aff1C[0  , 0] := 1.00000E+01; aff1C[0  , 1] := -4.03481E+00;
aff1C[1  , 0] := 1.99800E+01; aff1C[1  , 1] := -3.16200E+00;
aff1C[2  , 0] := 2.99600E+01; aff1C[2  , 1] := -2.64479E+00;
aff1C[3  , 0] := 3.99400E+01; aff1C[3  , 1] := -2.31488E+00;
aff1C[4  , 0] := 4.99200E+01; aff1C[4  , 1] := -2.09732E+00;
aff1C[5  , 0] := 5.99000E+01; aff1C[5  , 1] := -1.95840E+00;
aff1C[6  , 0] := 6.98800E+01; aff1C[6  , 1] := -1.87113E+00;
aff1C[7  , 0] := 7.98600E+01; aff1C[7  , 1] := -1.81732E+00;
aff1C[8  , 0] := 8.98400E+01; aff1C[8  , 1] := -1.78617E+00;
aff1C[9  , 0] := 9.98200E+01; aff1C[9  , 1] := -1.77164E+00;
aff1C[10 , 0] := 1.09800E+02; aff1C[10 , 1] := -1.76959E+00;
aff1C[11 , 0] := 1.19780E+02; aff1C[11 , 1] := -1.77729E+00;
aff1C[12 , 0] := 1.29760E+02; aff1C[12 , 1] := -1.79375E+00;
aff1C[13 , 0] := 1.39740E+02; aff1C[13 , 1] := -1.81862E+00;
aff1C[14 , 0] := 1.49720E+02; aff1C[14 , 1] := -1.85102E+00;
aff1C[15 , 0] := 1.59700E+02; aff1C[15 , 1] := -1.89079E+00;
aff1C[16 , 0] := 1.69680E+02; aff1C[16 , 1] := -1.93825E+00;
aff1C[17 , 0] := 1.79660E+02; aff1C[17 , 1] := -1.99421E+00;
aff1C[18 , 0] := 1.89640E+02; aff1C[18 , 1] := -2.05996E+00;
aff1C[19 , 0] := 1.99620E+02; aff1C[19 , 1] := -2.13743E+00;
aff1C[20 , 0] := 2.09600E+02; aff1C[20 , 1] := -2.22948E+00;
aff1C[21 , 0] := 2.19580E+02; aff1C[21 , 1] := -2.34037E+00;
aff1C[22 , 0] := 2.29560E+02; aff1C[22 , 1] := -2.47673E+00;
aff1C[23 , 0] := 2.39540E+02; aff1C[23 , 1] := -2.64947E+00;
aff1C[24 , 0] := 2.49520E+02; aff1C[24 , 1] := -2.87833E+00;
aff1C[25 , 0] := 2.59500E+02; aff1C[25 , 1] := -3.20451E+00;
aff1C[26 , 0] := 2.69480E+02; aff1C[26 , 1] := -3.73879E+00;
aff1C[27 , 0] := 2.79460E+02; aff1C[27 , 1] := -5.04188E+00;
aff1C[28 , 0] := 2.89440E+02; aff1C[28 , 1] := -4.53653E+00;
aff1C[29 , 0] := 2.99420E+02; aff1C[29 , 1] := -3.20323E+00;
aff1C[30 , 0] := 3.09400E+02; aff1C[30 , 1] := -2.53148E+00;
aff1C[31 , 0] := 3.19380E+02; aff1C[31 , 1] := -2.07370E+00;
aff1C[32 , 0] := 3.29360E+02; aff1C[32 , 1] := -1.72635E+00;
aff1C[33 , 0] := 3.39340E+02; aff1C[33 , 1] := -1.44913E+00;
aff1C[34 , 0] := 3.49320E+02; aff1C[34 , 1] := -1.22093E+00;
aff1C[35 , 0] := 3.59300E+02; aff1C[35 , 1] := -1.02921E+00;
aff1C[36 , 0] := 3.69280E+02; aff1C[36 , 1] := -8.65802E-01;
aff1C[37 , 0] := 3.79260E+02; aff1C[37 , 1] := -7.25116E-01;
aff1C[38 , 0] := 3.89240E+02; aff1C[38 , 1] := -6.03050E-01;
aff1C[39 , 0] := 3.99220E+02; aff1C[39 , 1] := -4.96466E-01;
aff1C[40 , 0] := 4.09200E+02; aff1C[40 , 1] := -4.02926E-01;
aff1C[41 , 0] := 4.19180E+02; aff1C[41 , 1] := -3.20489E-01;
aff1C[42 , 0] := 4.29160E+02; aff1C[42 , 1] := -2.47581E-01;
aff1C[43 , 0] := 4.39140E+02; aff1C[43 , 1] := -1.82911E-01;
aff1C[44 , 0] := 4.49120E+02; aff1C[44 , 1] := -1.25405E-01;
aff1C[45 , 0] := 4.59100E+02; aff1C[45 , 1] := -7.41593E-02;
aff1C[46 , 0] := 4.69080E+02; aff1C[46 , 1] := -2.84093E-02;
aff1C[47 , 0] := 4.79060E+02; aff1C[47 , 1] := 1.24973E-02;
aff1C[48 , 0] := 4.89040E+02; aff1C[48 , 1] := 4.91208E-02;
aff1C[49 , 0] := 4.99020E+02; aff1C[49 , 1] := 8.19448E-02;
aff1C[50 , 0] := 5.09000E+02; aff1C[50 , 1] := 1.11389E-01;
aff1C[51 , 0] := 5.18980E+02; aff1C[51 , 1] := 1.37819E-01;
aff1C[52 , 0] := 5.28960E+02; aff1C[52 , 1] := 1.61554E-01;
aff1C[53 , 0] := 5.38940E+02; aff1C[53 , 1] := 1.82875E-01;
aff1C[54 , 0] := 5.48920E+02; aff1C[54 , 1] := 2.02029E-01;
aff1C[55 , 0] := 5.58900E+02; aff1C[55 , 1] := 2.19234E-01;
aff1C[56 , 0] := 5.68880E+02; aff1C[56 , 1] := 2.34684E-01;
aff1C[57 , 0] := 5.78860E+02; aff1C[57 , 1] := 2.48550E-01;
aff1C[58 , 0] := 5.88840E+02; aff1C[58 , 1] := 2.60984E-01;
aff1C[59 , 0] := 5.98820E+02; aff1C[59 , 1] := 2.72123E-01;
aff1C[60 , 0] := 6.08800E+02; aff1C[60 , 1] := 2.82088E-01;
aff1C[61 , 0] := 6.18780E+02; aff1C[61 , 1] := 2.90989E-01;
aff1C[62 , 0] := 6.28760E+02; aff1C[62 , 1] := 2.98923E-01;
aff1C[63 , 0] := 6.38740E+02; aff1C[63 , 1] := 3.05978E-01;
aff1C[64 , 0] := 6.48720E+02; aff1C[64 , 1] := 3.12234E-01;
aff1C[65 , 0] := 6.58700E+02; aff1C[65 , 1] := 3.17761E-01;
aff1C[66 , 0] := 6.68680E+02; aff1C[66 , 1] := 3.22624E-01;
aff1C[67 , 0] := 6.78660E+02; aff1C[67 , 1] := 3.26882E-01;
aff1C[68 , 0] := 6.88640E+02; aff1C[68 , 1] := 3.30587E-01;
aff1C[69 , 0] := 6.98620E+02; aff1C[69 , 1] := 3.33787E-01;
aff1C[70 , 0] := 7.08600E+02; aff1C[70 , 1] := 3.36525E-01;
aff1C[71 , 0] := 7.18580E+02; aff1C[71 , 1] := 3.38842E-01;
aff1C[72 , 0] := 7.28560E+02; aff1C[72 , 1] := 3.40773E-01;
aff1C[73 , 0] := 7.38540E+02; aff1C[73 , 1] := 3.42351E-01;
aff1C[74 , 0] := 7.48520E+02; aff1C[74 , 1] := 3.43606E-01;
aff1C[75 , 0] := 7.58500E+02; aff1C[75 , 1] := 3.44565E-01;
aff1C[76 , 0] := 7.68480E+02; aff1C[76 , 1] := 3.45254E-01;
aff1C[77 , 0] := 7.78460E+02; aff1C[77 , 1] := 3.45694E-01;
aff1C[78 , 0] := 7.88440E+02; aff1C[78 , 1] := 3.45908E-01;
aff1C[79 , 0] := 7.98420E+02; aff1C[79 , 1] := 3.45914E-01;
aff1C[80 , 0] := 8.08400E+02; aff1C[80 , 1] := 3.45729E-01;
aff1C[81 , 0] := 8.18380E+02; aff1C[81 , 1] := 3.45371E-01;
aff1C[82 , 0] := 8.28360E+02; aff1C[82 , 1] := 3.44854E-01;
aff1C[83 , 0] := 8.38340E+02; aff1C[83 , 1] := 3.44196E-01;
aff1C[84 , 0] := 8.48320E+02; aff1C[84 , 1] := 3.43361E-01;
aff1C[85 , 0] := 8.58300E+02; aff1C[85 , 1] := 3.42839E-01;
aff1C[86 , 0] := 8.68280E+02; aff1C[86 , 1] := 3.41862E-01;
aff1C[87 , 0] := 8.78260E+02; aff1C[87 , 1] := 3.40748E-01;
aff1C[88 , 0] := 8.88240E+02; aff1C[88 , 1] := 3.39538E-01;
aff1C[89 , 0] := 8.98220E+02; aff1C[89 , 1] := 3.38248E-01;
aff1C[90 , 0] := 9.08200E+02; aff1C[90 , 1] := 3.36883E-01;
aff1C[91 , 0] := 9.18180E+02; aff1C[91 , 1] := 3.35451E-01;
aff1C[92 , 0] := 9.28160E+02; aff1C[92 , 1] := 3.33958E-01;
aff1C[93 , 0] := 9.38140E+02; aff1C[93 , 1] := 3.32411E-01;
aff1C[94 , 0] := 9.48120E+02; aff1C[94 , 1] := 3.30816E-01;
aff1C[95 , 0] := 9.58100E+02; aff1C[95 , 1] := 3.29178E-01;
aff1C[96 , 0] := 9.68080E+02; aff1C[96 , 1] := 3.27503E-01;
aff1C[97 , 0] := 9.78060E+02; aff1C[97 , 1] := 3.25794E-01;
aff1C[98 , 0] := 9.88040E+02; aff1C[98 , 1] := 3.24057E-01;
aff1C[99 , 0] := 9.98020E+02; aff1C[99 , 1] := 3.22295E-01;
aff1C[100, 0] := 1.00800E+03; aff1C[100, 1] := 3.20475E-01;
aff1C[101, 0] := 1.01798E+03; aff1C[101, 1] := 3.18626E-01;
aff1C[102, 0] := 1.02796E+03; aff1C[102, 1] := 3.16761E-01;
aff1C[103, 0] := 1.03794E+03; aff1C[103, 1] := 3.14881E-01;
aff1C[104, 0] := 1.04792E+03; aff1C[104, 1] := 3.12989E-01;
aff1C[105, 0] := 1.05790E+03; aff1C[105, 1] := 3.11086E-01;
aff1C[106, 0] := 1.06788E+03; aff1C[106, 1] := 3.09176E-01;
aff1C[107, 0] := 1.07786E+03; aff1C[107, 1] := 3.07262E-01;
aff1C[108, 0] := 1.08784E+03; aff1C[108, 1] := 3.05346E-01;
aff1C[109, 0] := 1.09782E+03; aff1C[109, 1] := 3.03433E-01;
aff1C[110, 0] := 1.10780E+03; aff1C[110, 1] := 3.01524E-01;
aff1C[111, 0] := 1.11778E+03; aff1C[111, 1] := 2.99623E-01;
aff1C[112, 0] := 1.12776E+03; aff1C[112, 1] := 2.97736E-01;
aff1C[113, 0] := 1.13774E+03; aff1C[113, 1] := 2.95857E-01;
aff1C[114, 0] := 1.14772E+03; aff1C[114, 1] := 2.93954E-01;
aff1C[115, 0] := 1.15770E+03; aff1C[115, 1] := 2.92011E-01;
aff1C[116, 0] := 1.16768E+03; aff1C[116, 1] := 2.90036E-01;
aff1C[117, 0] := 1.17766E+03; aff1C[117, 1] := 2.88036E-01;
aff1C[118, 0] := 1.18764E+03; aff1C[118, 1] := 2.86016E-01;
aff1C[119, 0] := 1.19762E+03; aff1C[119, 1] := 2.83981E-01;
aff1C[120, 0] := 1.20760E+03; aff1C[120, 1] := 2.81934E-01;
aff1C[121, 0] := 1.21758E+03; aff1C[121, 1] := 2.79880E-01;
aff1C[122, 0] := 1.22756E+03; aff1C[122, 1] := 2.77820E-01;
aff1C[123, 0] := 1.23754E+03; aff1C[123, 1] := 2.75758E-01;
aff1C[124, 0] := 1.24752E+03; aff1C[124, 1] := 2.73697E-01;
aff1C[125, 0] := 1.25750E+03; aff1C[125, 1] := 2.71637E-01;
aff1C[126, 0] := 1.26748E+03; aff1C[126, 1] := 2.69581E-01;
aff1C[127, 0] := 1.27746E+03; aff1C[127, 1] := 2.67530E-01;
aff1C[128, 0] := 1.28744E+03; aff1C[128, 1] := 2.65487E-01;
aff1C[129, 0] := 1.29742E+03; aff1C[129, 1] := 2.63451E-01;
aff1C[130, 0] := 1.30740E+03; aff1C[130, 1] := 2.61425E-01;
aff1C[131, 0] := 1.31738E+03; aff1C[131, 1] := 2.59409E-01;
aff1C[132, 0] := 1.32736E+03; aff1C[132, 1] := 2.57404E-01;
aff1C[133, 0] := 1.33734E+03; aff1C[133, 1] := 2.55410E-01;
aff1C[134, 0] := 1.34732E+03; aff1C[134, 1] := 2.53430E-01;
aff1C[135, 0] := 1.35730E+03; aff1C[135, 1] := 2.51462E-01;
aff1C[136, 0] := 1.36728E+03; aff1C[136, 1] := 2.49508E-01;
aff1C[137, 0] := 1.37726E+03; aff1C[137, 1] := 2.47568E-01;
aff1C[138, 0] := 1.38724E+03; aff1C[138, 1] := 2.45643E-01;
aff1C[139, 0] := 1.39722E+03; aff1C[139, 1] := 2.43732E-01;
aff1C[140, 0] := 1.40720E+03; aff1C[140, 1] := 2.41837E-01;
aff1C[141, 0] := 1.41718E+03; aff1C[141, 1] := 2.39957E-01;
aff1C[142, 0] := 1.42716E+03; aff1C[142, 1] := 2.38093E-01;
aff1C[143, 0] := 1.43714E+03; aff1C[143, 1] := 2.36244E-01;
aff1C[144, 0] := 1.44712E+03; aff1C[144, 1] := 2.34412E-01;
aff1C[145, 0] := 1.45710E+03; aff1C[145, 1] := 2.32596E-01;
aff1C[146, 0] := 1.46708E+03; aff1C[146, 1] := 2.30796E-01;
aff1C[147, 0] := 1.47706E+03; aff1C[147, 1] := 2.29012E-01;
aff1C[148, 0] := 1.48704E+03; aff1C[148, 1] := 2.27245E-01;
aff1C[149, 0] := 1.49702E+03; aff1C[149, 1] := 2.25494E-01;
aff1C[150, 0] := 1.50700E+03; aff1C[150, 1] := 2.23759E-01;
aff1C[151, 0] := 1.51698E+03; aff1C[151, 1] := 2.22041E-01;
aff1C[152, 0] := 1.52696E+03; aff1C[152, 1] := 2.20340E-01;
aff1C[153, 0] := 1.53694E+03; aff1C[153, 1] := 2.18655E-01;
aff1C[154, 0] := 1.54692E+03; aff1C[154, 1] := 2.16986E-01;
aff1C[155, 0] := 1.55690E+03; aff1C[155, 1] := 2.15333E-01;
aff1C[156, 0] := 1.56688E+03; aff1C[156, 1] := 2.13697E-01;
aff1C[157, 0] := 1.57686E+03; aff1C[157, 1] := 2.12077E-01;
aff1C[158, 0] := 1.58684E+03; aff1C[158, 1] := 2.10473E-01;
aff1C[159, 0] := 1.59682E+03; aff1C[159, 1] := 2.08884E-01;
aff1C[160, 0] := 1.60680E+03; aff1C[160, 1] := 2.07312E-01;
aff1C[161, 0] := 1.61678E+03; aff1C[161, 1] := 2.05756E-01;
aff1C[162, 0] := 1.62676E+03; aff1C[162, 1] := 2.04215E-01;
aff1C[163, 0] := 1.63674E+03; aff1C[163, 1] := 2.02690E-01;
aff1C[164, 0] := 1.64672E+03; aff1C[164, 1] := 2.01180E-01;
aff1C[165, 0] := 1.65670E+03; aff1C[165, 1] := 1.99686E-01;
aff1C[166, 0] := 1.66668E+03; aff1C[166, 1] := 1.98206E-01;
aff1C[167, 0] := 1.67666E+03; aff1C[167, 1] := 1.96742E-01;
aff1C[168, 0] := 1.68664E+03; aff1C[168, 1] := 1.95293E-01;
aff1C[169, 0] := 1.69662E+03; aff1C[169, 1] := 1.93859E-01;
aff1C[170, 0] := 1.70660E+03; aff1C[170, 1] := 1.92439E-01;
aff1C[171, 0] := 1.71658E+03; aff1C[171, 1] := 1.91034E-01;
aff1C[172, 0] := 1.72656E+03; aff1C[172, 1] := 1.89643E-01;
aff1C[173, 0] := 1.73654E+03; aff1C[173, 1] := 1.88266E-01;
aff1C[174, 0] := 1.74652E+03; aff1C[174, 1] := 1.86904E-01;
aff1C[175, 0] := 1.75650E+03; aff1C[175, 1] := 1.85555E-01;
aff1C[176, 0] := 1.76648E+03; aff1C[176, 1] := 1.84221E-01;
aff1C[177, 0] := 1.77646E+03; aff1C[177, 1] := 1.82900E-01;
aff1C[178, 0] := 1.78644E+03; aff1C[178, 1] := 1.81592E-01;
aff1C[179, 0] := 1.79642E+03; aff1C[179, 1] := 1.80298E-01;
aff1C[180, 0] := 1.80640E+03; aff1C[180, 1] := 1.79018E-01;
aff1C[181, 0] := 1.81638E+03; aff1C[181, 1] := 1.77750E-01;
aff1C[182, 0] := 1.82636E+03; aff1C[182, 1] := 1.76495E-01;
aff1C[183, 0] := 1.83634E+03; aff1C[183, 1] := 1.75254E-01;
aff1C[184, 0] := 1.84632E+03; aff1C[184, 1] := 1.74024E-01;
aff1C[185, 0] := 1.85630E+03; aff1C[185, 1] := 1.72808E-01;
aff1C[186, 0] := 1.86628E+03; aff1C[186, 1] := 1.71604E-01;
aff1C[187, 0] := 1.87626E+03; aff1C[187, 1] := 1.70412E-01;
aff1C[188, 0] := 1.88624E+03; aff1C[188, 1] := 1.69232E-01;
aff1C[189, 0] := 1.89622E+03; aff1C[189, 1] := 1.68064E-01;
aff1C[190, 0] := 1.90620E+03; aff1C[190, 1] := 1.66908E-01;
aff1C[191, 0] := 1.91618E+03; aff1C[191, 1] := 1.65764E-01;
aff1C[192, 0] := 1.92616E+03; aff1C[192, 1] := 1.64631E-01;
aff1C[193, 0] := 1.93614E+03; aff1C[193, 1] := 1.63510E-01;
aff1C[194, 0] := 1.94612E+03; aff1C[194, 1] := 1.62400E-01;
aff1C[195, 0] := 1.95610E+03; aff1C[195, 1] := 1.61301E-01;
aff1C[196, 0] := 1.96608E+03; aff1C[196, 1] := 1.60214E-01;
aff1C[197, 0] := 1.97606E+03; aff1C[197, 1] := 1.59137E-01;
aff1C[198, 0] := 1.98604E+03; aff1C[198, 1] := 1.58071E-01;
aff1C[199, 0] := 1.99602E+03; aff1C[199, 1] := 1.57015E-01;
aff1C[200, 0] := 2.00600E+03; aff1C[200, 1] := 1.55971E-01;
aff1C[201, 0] := 2.01598E+03; aff1C[201, 1] := 1.54936E-01;
aff1C[202, 0] := 2.02596E+03; aff1C[202, 1] := 1.53912E-01;
aff1C[203, 0] := 2.03594E+03; aff1C[203, 1] := 1.52898E-01;
aff1C[204, 0] := 2.04592E+03; aff1C[204, 1] := 1.51894E-01;
aff1C[205, 0] := 2.05590E+03; aff1C[205, 1] := 1.50900E-01;
aff1C[206, 0] := 2.06588E+03; aff1C[206, 1] := 1.49916E-01;
aff1C[207, 0] := 2.07586E+03; aff1C[207, 1] := 1.48942E-01;
aff1C[208, 0] := 2.08584E+03; aff1C[208, 1] := 1.47977E-01;
aff1C[209, 0] := 2.09582E+03; aff1C[209, 1] := 1.47022E-01;
aff1C[210, 0] := 2.10580E+03; aff1C[210, 1] := 1.46076E-01;
aff1C[211, 0] := 2.11578E+03; aff1C[211, 1] := 1.45139E-01;
aff1C[212, 0] := 2.12576E+03; aff1C[212, 1] := 1.44211E-01;
aff1C[213, 0] := 2.13574E+03; aff1C[213, 1] := 1.43292E-01;
aff1C[214, 0] := 2.14572E+03; aff1C[214, 1] := 1.42383E-01;
aff1C[215, 0] := 2.15570E+03; aff1C[215, 1] := 1.41482E-01;
aff1C[216, 0] := 2.16568E+03; aff1C[216, 1] := 1.40590E-01;
aff1C[217, 0] := 2.17566E+03; aff1C[217, 1] := 1.39706E-01;
aff1C[218, 0] := 2.18564E+03; aff1C[218, 1] := 1.38831E-01;
aff1C[219, 0] := 2.19562E+03; aff1C[219, 1] := 1.37964E-01;
aff1C[220, 0] := 2.20560E+03; aff1C[220, 1] := 1.37106E-01;
aff1C[221, 0] := 2.21558E+03; aff1C[221, 1] := 1.36256E-01;
aff1C[222, 0] := 2.22556E+03; aff1C[222, 1] := 1.35414E-01;
aff1C[223, 0] := 2.23554E+03; aff1C[223, 1] := 1.34580E-01;
aff1C[224, 0] := 2.24552E+03; aff1C[224, 1] := 1.33753E-01;
aff1C[225, 0] := 2.25550E+03; aff1C[225, 1] := 1.32935E-01;
aff1C[226, 0] := 2.26548E+03; aff1C[226, 1] := 1.32125E-01;
aff1C[227, 0] := 2.27546E+03; aff1C[227, 1] := 1.31322E-01;
aff1C[228, 0] := 2.28544E+03; aff1C[228, 1] := 1.30526E-01;
aff1C[229, 0] := 2.29542E+03; aff1C[229, 1] := 1.29739E-01;
aff1C[230, 0] := 2.30540E+03; aff1C[230, 1] := 1.28958E-01;
aff1C[231, 0] := 2.31538E+03; aff1C[231, 1] := 1.28185E-01;
aff1C[232, 0] := 2.32536E+03; aff1C[232, 1] := 1.27419E-01;
aff1C[233, 0] := 2.33534E+03; aff1C[233, 1] := 1.26660E-01;
aff1C[234, 0] := 2.34532E+03; aff1C[234, 1] := 1.25908E-01;
aff1C[235, 0] := 2.35530E+03; aff1C[235, 1] := 1.25164E-01;
aff1C[236, 0] := 2.36528E+03; aff1C[236, 1] := 1.24426E-01;
aff1C[237, 0] := 2.37526E+03; aff1C[237, 1] := 1.23695E-01;
aff1C[238, 0] := 2.38524E+03; aff1C[238, 1] := 1.22970E-01;
aff1C[239, 0] := 2.39522E+03; aff1C[239, 1] := 1.22253E-01;
aff1C[240, 0] := 2.40520E+03; aff1C[240, 1] := 1.21541E-01;
aff1C[241, 0] := 2.41518E+03; aff1C[241, 1] := 1.20837E-01;
aff1C[242, 0] := 2.42516E+03; aff1C[242, 1] := 1.20139E-01;
aff1C[243, 0] := 2.43514E+03; aff1C[243, 1] := 1.19447E-01;
aff1C[244, 0] := 2.44512E+03; aff1C[244, 1] := 1.18761E-01;
aff1C[245, 0] := 2.45510E+03; aff1C[245, 1] := 1.18082E-01;
aff1C[246, 0] := 2.46508E+03; aff1C[246, 1] := 1.17409E-01;
aff1C[247, 0] := 2.47506E+03; aff1C[247, 1] := 1.16742E-01;
aff1C[248, 0] := 2.48504E+03; aff1C[248, 1] := 1.16081E-01;
aff1C[249, 0] := 2.49502E+03; aff1C[249, 1] := 1.15426E-01;
aff1C[250, 0] := 2.50500E+03; aff1C[250, 1] := 1.14777E-01;
aff1C[251, 0] := 2.51498E+03; aff1C[251, 1] := 1.14134E-01;
aff1C[252, 0] := 2.52496E+03; aff1C[252, 1] := 1.13496E-01;
aff1C[253, 0] := 2.53494E+03; aff1C[253, 1] := 1.12864E-01;
aff1C[254, 0] := 2.54492E+03; aff1C[254, 1] := 1.12238E-01;
aff1C[255, 0] := 2.55490E+03; aff1C[255, 1] := 1.11617E-01;
aff1C[256, 0] := 2.56488E+03; aff1C[256, 1] := 1.11002E-01;
aff1C[257, 0] := 2.57486E+03; aff1C[257, 1] := 1.10393E-01;
aff1C[258, 0] := 2.58484E+03; aff1C[258, 1] := 1.09789E-01;
aff1C[259, 0] := 2.59482E+03; aff1C[259, 1] := 1.09190E-01;
aff1C[260, 0] := 2.60480E+03; aff1C[260, 1] := 1.08596E-01;
aff1C[261, 0] := 2.61478E+03; aff1C[261, 1] := 1.08008E-01;
aff1C[262, 0] := 2.62476E+03; aff1C[262, 1] := 1.07425E-01;
aff1C[263, 0] := 2.63474E+03; aff1C[263, 1] := 1.06847E-01;
aff1C[264, 0] := 2.64472E+03; aff1C[264, 1] := 1.06274E-01;
aff1C[265, 0] := 2.65470E+03; aff1C[265, 1] := 1.05706E-01;
aff1C[266, 0] := 2.66468E+03; aff1C[266, 1] := 1.05143E-01;
aff1C[267, 0] := 2.67466E+03; aff1C[267, 1] := 1.04585E-01;
aff1C[268, 0] := 2.68464E+03; aff1C[268, 1] := 1.04032E-01;
aff1C[269, 0] := 2.69462E+03; aff1C[269, 1] := 1.03484E-01;
aff1C[270, 0] := 2.70460E+03; aff1C[270, 1] := 1.02940E-01;
aff1C[271, 0] := 2.71458E+03; aff1C[271, 1] := 1.02402E-01;
aff1C[272, 0] := 2.72456E+03; aff1C[272, 1] := 1.01868E-01;
aff1C[273, 0] := 2.73454E+03; aff1C[273, 1] := 1.01338E-01;
aff1C[274, 0] := 2.74452E+03; aff1C[274, 1] := 1.00813E-01;
aff1C[275, 0] := 2.75450E+03; aff1C[275, 1] := 1.00293E-01;
aff1C[276, 0] := 2.76448E+03; aff1C[276, 1] := 9.97774E-02;
aff1C[277, 0] := 2.77446E+03; aff1C[277, 1] := 9.92662E-02;
aff1C[278, 0] := 2.78444E+03; aff1C[278, 1] := 9.87594E-02;
aff1C[279, 0] := 2.79442E+03; aff1C[279, 1] := 9.82570E-02;
aff1C[280, 0] := 2.80440E+03; aff1C[280, 1] := 9.77590E-02;
aff1C[281, 0] := 2.81438E+03; aff1C[281, 1] := 9.72652E-02;
aff1C[282, 0] := 2.82436E+03; aff1C[282, 1] := 9.67758E-02;
aff1C[283, 0] := 2.83434E+03; aff1C[283, 1] := 9.62906E-02;
aff1C[284, 0] := 2.84432E+03; aff1C[284, 1] := 9.58096E-02;
aff1C[285, 0] := 2.85430E+03; aff1C[285, 1] := 9.53328E-02;
aff1C[286, 0] := 2.86428E+03; aff1C[286, 1] := 9.48602E-02;
aff1C[287, 0] := 2.87426E+03; aff1C[287, 1] := 9.43916E-02;
aff1C[288, 0] := 2.88424E+03; aff1C[288, 1] := 9.39271E-02;
aff1C[289, 0] := 2.89422E+03; aff1C[289, 1] := 9.34666E-02;
aff1C[290, 0] := 2.90420E+03; aff1C[290, 1] := 9.30102E-02;
aff1C[291, 0] := 2.91418E+03; aff1C[291, 1] := 9.25577E-02;
aff1C[292, 0] := 2.92416E+03; aff1C[292, 1] := 9.21092E-02;
aff1C[293, 0] := 2.93414E+03; aff1C[293, 1] := 9.16645E-02;
aff1C[294, 0] := 2.94412E+03; aff1C[294, 1] := 9.12237E-02;
aff1C[295, 0] := 2.95410E+03; aff1C[295, 1] := 9.07871E-02;
aff1C[296, 0] := 2.96408E+03; aff1C[296, 1] := 9.03545E-02;
aff1C[297, 0] := 2.97406E+03; aff1C[297, 1] := 8.99253E-02;
aff1C[298, 0] := 2.98404E+03; aff1C[298, 1] := 8.94991E-02;
aff1C[299, 0] := 2.99402E+03; aff1C[299, 1] := 8.90753E-02;
aff1C[300, 0] := 3.00400E+03; aff1C[300, 1] := 8.86529E-02;
aff1C[301, 0] := 3.01398E+03; aff1C[301, 1] := 8.82307E-02;
aff1C[302, 0] := 3.02396E+03; aff1C[302, 1] := 8.78083E-02;
aff1C[303, 0] := 3.03394E+03; aff1C[303, 1] := 8.73870E-02;
aff1C[304, 0] := 3.04392E+03; aff1C[304, 1] := 8.69680E-02;
aff1C[305, 0] := 3.05390E+03; aff1C[305, 1] := 8.65522E-02;
aff1C[306, 0] := 3.06388E+03; aff1C[306, 1] := 8.61393E-02;
aff1C[307, 0] := 3.07386E+03; aff1C[307, 1] := 8.57290E-02;
aff1C[308, 0] := 3.08384E+03; aff1C[308, 1] := 8.53210E-02;
aff1C[309, 0] := 3.09382E+03; aff1C[309, 1] := 8.49154E-02;
aff1C[310, 0] := 3.10380E+03; aff1C[310, 1] := 8.45123E-02;
aff1C[311, 0] := 3.11378E+03; aff1C[311, 1] := 8.41118E-02;
aff1C[312, 0] := 3.12376E+03; aff1C[312, 1] := 8.37137E-02;
aff1C[313, 0] := 3.13374E+03; aff1C[313, 1] := 8.33180E-02;
aff1C[314, 0] := 3.14372E+03; aff1C[314, 1] := 8.29248E-02;
aff1C[315, 0] := 3.15370E+03; aff1C[315, 1] := 8.25341E-02;
aff1C[316, 0] := 3.16368E+03; aff1C[316, 1] := 8.21458E-02;
aff1C[317, 0] := 3.17366E+03; aff1C[317, 1] := 8.17599E-02;
aff1C[318, 0] := 3.18364E+03; aff1C[318, 1] := 8.13764E-02;
aff1C[319, 0] := 3.19362E+03; aff1C[319, 1] := 8.09953E-02;
aff1C[320, 0] := 3.20360E+03; aff1C[320, 1] := 8.06166E-02;
aff1C[321, 0] := 3.21358E+03; aff1C[321, 1] := 8.02403E-02;
aff1C[322, 0] := 3.22356E+03; aff1C[322, 1] := 7.98663E-02;
aff1C[323, 0] := 3.23354E+03; aff1C[323, 1] := 7.94947E-02;
aff1C[324, 0] := 3.24352E+03; aff1C[324, 1] := 7.91254E-02;
aff1C[325, 0] := 3.25350E+03; aff1C[325, 1] := 7.87584E-02;
aff1C[326, 0] := 3.26348E+03; aff1C[326, 1] := 7.83938E-02;
aff1C[327, 0] := 3.27346E+03; aff1C[327, 1] := 7.80314E-02;
aff1C[328, 0] := 3.28344E+03; aff1C[328, 1] := 7.76714E-02;
aff1C[329, 0] := 3.29342E+03; aff1C[329, 1] := 7.73136E-02;
aff1C[330, 0] := 3.30340E+03; aff1C[330, 1] := 7.69580E-02;
aff1C[331, 0] := 3.31338E+03; aff1C[331, 1] := 7.66047E-02;
aff1C[332, 0] := 3.32336E+03; aff1C[332, 1] := 7.62536E-02;
aff1C[333, 0] := 3.33334E+03; aff1C[333, 1] := 7.59048E-02;
aff1C[334, 0] := 3.34332E+03; aff1C[334, 1] := 7.55581E-02;
aff1C[335, 0] := 3.35330E+03; aff1C[335, 1] := 7.52136E-02;
aff1C[336, 0] := 3.36328E+03; aff1C[336, 1] := 7.48713E-02;
aff1C[337, 0] := 3.37326E+03; aff1C[337, 1] := 7.45311E-02;
aff1C[338, 0] := 3.38324E+03; aff1C[338, 1] := 7.41931E-02;
aff1C[339, 0] := 3.39322E+03; aff1C[339, 1] := 7.38572E-02;
aff1C[340, 0] := 3.40320E+03; aff1C[340, 1] := 7.35234E-02;
aff1C[341, 0] := 3.41318E+03; aff1C[341, 1] := 7.31918E-02;
aff1C[342, 0] := 3.42316E+03; aff1C[342, 1] := 7.28622E-02;
aff1C[343, 0] := 3.43314E+03; aff1C[343, 1] := 7.25346E-02;
aff1C[344, 0] := 3.44312E+03; aff1C[344, 1] := 7.22092E-02;
aff1C[345, 0] := 3.45310E+03; aff1C[345, 1] := 7.18857E-02;
aff1C[346, 0] := 3.46308E+03; aff1C[346, 1] := 7.15643E-02;
aff1C[347, 0] := 3.47306E+03; aff1C[347, 1] := 7.12450E-02;
aff1C[348, 0] := 3.48304E+03; aff1C[348, 1] := 7.09276E-02;
aff1C[349, 0] := 3.49302E+03; aff1C[349, 1] := 7.06122E-02;
aff1C[350, 0] := 3.50300E+03; aff1C[350, 1] := 7.02987E-02;
aff1C[351, 0] := 3.51298E+03; aff1C[351, 1] := 6.99873E-02;
aff1C[352, 0] := 3.52296E+03; aff1C[352, 1] := 6.96777E-02;
aff1C[353, 0] := 3.53294E+03; aff1C[353, 1] := 6.93701E-02;
aff1C[354, 0] := 3.54292E+03; aff1C[354, 1] := 6.90645E-02;
aff1C[355, 0] := 3.55290E+03; aff1C[355, 1] := 6.87607E-02;
aff1C[356, 0] := 3.56288E+03; aff1C[356, 1] := 6.84588E-02;
aff1C[357, 0] := 3.57286E+03; aff1C[357, 1] := 6.81587E-02;
aff1C[358, 0] := 3.58284E+03; aff1C[358, 1] := 6.78606E-02;
aff1C[359, 0] := 3.59282E+03; aff1C[359, 1] := 6.75642E-02;
aff1C[360, 0] := 3.60280E+03; aff1C[360, 1] := 6.72698E-02;
aff1C[361, 0] := 3.61278E+03; aff1C[361, 1] := 6.69771E-02;
aff1C[362, 0] := 3.62276E+03; aff1C[362, 1] := 6.66862E-02;
aff1C[363, 0] := 3.63274E+03; aff1C[363, 1] := 6.63972E-02;
aff1C[364, 0] := 3.64272E+03; aff1C[364, 1] := 6.61099E-02;
aff1C[365, 0] := 3.65270E+03; aff1C[365, 1] := 6.58243E-02;
aff1C[366, 0] := 3.66268E+03; aff1C[366, 1] := 6.55406E-02;
aff1C[367, 0] := 3.67266E+03; aff1C[367, 1] := 6.52585E-02;
aff1C[368, 0] := 3.68264E+03; aff1C[368, 1] := 6.49782E-02;
aff1C[369, 0] := 3.69262E+03; aff1C[369, 1] := 6.46996E-02;
aff1C[370, 0] := 3.70260E+03; aff1C[370, 1] := 6.44228E-02;
aff1C[371, 0] := 3.71258E+03; aff1C[371, 1] := 6.41476E-02;
aff1C[372, 0] := 3.72256E+03; aff1C[372, 1] := 6.38740E-02;
aff1C[373, 0] := 3.73254E+03; aff1C[373, 1] := 6.36022E-02;
aff1C[374, 0] := 3.74252E+03; aff1C[374, 1] := 6.33320E-02;
aff1C[375, 0] := 3.75250E+03; aff1C[375, 1] := 6.30634E-02;
aff1C[376, 0] := 3.76248E+03; aff1C[376, 1] := 6.27965E-02;
aff1C[377, 0] := 3.77246E+03; aff1C[377, 1] := 6.25311E-02;
aff1C[378, 0] := 3.78244E+03; aff1C[378, 1] := 6.22674E-02;
aff1C[379, 0] := 3.79242E+03; aff1C[379, 1] := 6.20053E-02;
aff1C[380, 0] := 3.80240E+03; aff1C[380, 1] := 6.17447E-02;
aff1C[381, 0] := 3.81238E+03; aff1C[381, 1] := 6.14858E-02;
aff1C[382, 0] := 3.82236E+03; aff1C[382, 1] := 6.12283E-02;
aff1C[383, 0] := 3.83234E+03; aff1C[383, 1] := 6.09724E-02;
aff1C[384, 0] := 3.84232E+03; aff1C[384, 1] := 6.07181E-02;
aff1C[385, 0] := 3.85230E+03; aff1C[385, 1] := 6.04653E-02;
aff1C[386, 0] := 3.86228E+03; aff1C[386, 1] := 6.02139E-02;
aff1C[387, 0] := 3.87226E+03; aff1C[387, 1] := 5.99641E-02;
aff1C[388, 0] := 3.88224E+03; aff1C[388, 1] := 5.97158E-02;
aff1C[389, 0] := 3.89222E+03; aff1C[389, 1] := 5.94689E-02;
aff1C[390, 0] := 3.90220E+03; aff1C[390, 1] := 5.92235E-02;
aff1C[391, 0] := 3.91218E+03; aff1C[391, 1] := 5.89796E-02;
aff1C[392, 0] := 3.92216E+03; aff1C[392, 1] := 5.87371E-02;
aff1C[393, 0] := 3.93214E+03; aff1C[393, 1] := 5.84960E-02;
aff1C[394, 0] := 3.94212E+03; aff1C[394, 1] := 5.82564E-02;
aff1C[395, 0] := 3.95210E+03; aff1C[395, 1] := 5.80182E-02;
aff1C[396, 0] := 3.96208E+03; aff1C[396, 1] := 5.77814E-02;
aff1C[397, 0] := 3.97206E+03; aff1C[397, 1] := 5.75459E-02;
aff1C[398, 0] := 3.98204E+03; aff1C[398, 1] := 5.73119E-02;
aff1C[399, 0] := 3.99202E+03; aff1C[399, 1] := 5.70792E-02;
aff1C[400, 0] := 4.00200E+03; aff1C[400, 1] := 5.68479E-02;
aff1C[401, 0] := 4.01198E+03; aff1C[401, 1] := 5.66179E-02;
aff1C[402, 0] := 4.02196E+03; aff1C[402, 1] := 5.63892E-02;
aff1C[403, 0] := 4.03194E+03; aff1C[403, 1] := 5.61619E-02;
aff1C[404, 0] := 4.04192E+03; aff1C[404, 1] := 5.59360E-02;
aff1C[405, 0] := 4.05190E+03; aff1C[405, 1] := 5.57113E-02;
aff1C[406, 0] := 4.06188E+03; aff1C[406, 1] := 5.54879E-02;
aff1C[407, 0] := 4.07186E+03; aff1C[407, 1] := 5.52658E-02;
aff1C[408, 0] := 4.08184E+03; aff1C[408, 1] := 5.50450E-02;
aff1C[409, 0] := 4.09182E+03; aff1C[409, 1] := 5.48255E-02;
aff1C[410, 0] := 4.10180E+03; aff1C[410, 1] := 5.46072E-02;
aff1C[411, 0] := 4.11178E+03; aff1C[411, 1] := 5.43902E-02;
aff1C[412, 0] := 4.12176E+03; aff1C[412, 1] := 5.41744E-02;
aff1C[413, 0] := 4.13174E+03; aff1C[413, 1] := 5.39599E-02;
aff1C[414, 0] := 4.14172E+03; aff1C[414, 1] := 5.37466E-02;
aff1C[415, 0] := 4.15170E+03; aff1C[415, 1] := 5.35345E-02;
aff1C[416, 0] := 4.16168E+03; aff1C[416, 1] := 5.33236E-02;
aff1C[417, 0] := 4.17166E+03; aff1C[417, 1] := 5.31139E-02;
aff1C[418, 0] := 4.18164E+03; aff1C[418, 1] := 5.29054E-02;
aff1C[419, 0] := 4.19162E+03; aff1C[419, 1] := 5.26981E-02;
aff1C[420, 0] := 4.20160E+03; aff1C[420, 1] := 5.24920E-02;
aff1C[421, 0] := 4.21158E+03; aff1C[421, 1] := 5.22870E-02;
aff1C[422, 0] := 4.22156E+03; aff1C[422, 1] := 5.20832E-02;
aff1C[423, 0] := 4.23154E+03; aff1C[423, 1] := 5.18805E-02;
aff1C[424, 0] := 4.24152E+03; aff1C[424, 1] := 5.16790E-02;
aff1C[425, 0] := 4.25150E+03; aff1C[425, 1] := 5.14786E-02;
aff1C[426, 0] := 4.26148E+03; aff1C[426, 1] := 5.12793E-02;
aff1C[427, 0] := 4.27146E+03; aff1C[427, 1] := 5.10812E-02;
aff1C[428, 0] := 4.28144E+03; aff1C[428, 1] := 5.08841E-02;
aff1C[429, 0] := 4.29142E+03; aff1C[429, 1] := 5.06882E-02;
aff1C[430, 0] := 4.30140E+03; aff1C[430, 1] := 5.04933E-02;
aff1C[431, 0] := 4.31138E+03; aff1C[431, 1] := 5.02995E-02;
aff1C[432, 0] := 4.32136E+03; aff1C[432, 1] := 5.01068E-02;
aff1C[433, 0] := 4.33134E+03; aff1C[433, 1] := 4.99152E-02;
aff1C[434, 0] := 4.34132E+03; aff1C[434, 1] := 4.97246E-02;
aff1C[435, 0] := 4.35130E+03; aff1C[435, 1] := 4.95351E-02;
aff1C[436, 0] := 4.36128E+03; aff1C[436, 1] := 4.93466E-02;
aff1C[437, 0] := 4.37126E+03; aff1C[437, 1] := 4.91592E-02;
aff1C[438, 0] := 4.38124E+03; aff1C[438, 1] := 4.89728E-02;
aff1C[439, 0] := 4.39122E+03; aff1C[439, 1] := 4.87874E-02;
aff1C[440, 0] := 4.40120E+03; aff1C[440, 1] := 4.86030E-02;
aff1C[441, 0] := 4.41118E+03; aff1C[441, 1] := 4.84197E-02;
aff1C[442, 0] := 4.42116E+03; aff1C[442, 1] := 4.82373E-02;
aff1C[443, 0] := 4.43114E+03; aff1C[443, 1] := 4.80560E-02;
aff1C[444, 0] := 4.44112E+03; aff1C[444, 1] := 4.78756E-02;
aff1C[445, 0] := 4.45110E+03; aff1C[445, 1] := 4.76962E-02;
aff1C[446, 0] := 4.46108E+03; aff1C[446, 1] := 4.75178E-02;
aff1C[447, 0] := 4.47106E+03; aff1C[447, 1] := 4.73403E-02;
aff1C[448, 0] := 4.48104E+03; aff1C[448, 1] := 4.71638E-02;
aff1C[449, 0] := 4.49102E+03; aff1C[449, 1] := 4.69883E-02;
aff1C[450, 0] := 4.50100E+03; aff1C[450, 1] := 4.68137E-02;
aff1C[451, 0] := 4.51098E+03; aff1C[451, 1] := 4.66400E-02;
aff1C[452, 0] := 4.52096E+03; aff1C[452, 1] := 4.64673E-02;
aff1C[453, 0] := 4.53094E+03; aff1C[453, 1] := 4.62955E-02;
aff1C[454, 0] := 4.54092E+03; aff1C[454, 1] := 4.61246E-02;
aff1C[455, 0] := 4.55090E+03; aff1C[455, 1] := 4.59547E-02;
aff1C[456, 0] := 4.56088E+03; aff1C[456, 1] := 4.57856E-02;
aff1C[457, 0] := 4.57086E+03; aff1C[457, 1] := 4.56175E-02;
aff1C[458, 0] := 4.58084E+03; aff1C[458, 1] := 4.54502E-02;
aff1C[459, 0] := 4.59082E+03; aff1C[459, 1] := 4.52838E-02;
aff1C[460, 0] := 4.60080E+03; aff1C[460, 1] := 4.51183E-02;
aff1C[461, 0] := 4.61078E+03; aff1C[461, 1] := 4.49537E-02;
aff1C[462, 0] := 4.62076E+03; aff1C[462, 1] := 4.47900E-02;
aff1C[463, 0] := 4.63074E+03; aff1C[463, 1] := 4.46271E-02;
aff1C[464, 0] := 4.64072E+03; aff1C[464, 1] := 4.44651E-02;
aff1C[465, 0] := 4.65070E+03; aff1C[465, 1] := 4.43040E-02;
aff1C[466, 0] := 4.66068E+03; aff1C[466, 1] := 4.41436E-02;
aff1C[467, 0] := 4.67066E+03; aff1C[467, 1] := 4.39842E-02;
aff1C[468, 0] := 4.68064E+03; aff1C[468, 1] := 4.38255E-02;
aff1C[469, 0] := 4.69062E+03; aff1C[469, 1] := 4.36677E-02;
aff1C[470, 0] := 4.70060E+03; aff1C[470, 1] := 4.35107E-02;
aff1C[471, 0] := 4.71058E+03; aff1C[471, 1] := 4.33546E-02;
aff1C[472, 0] := 4.72056E+03; aff1C[472, 1] := 4.31992E-02;
aff1C[473, 0] := 4.73054E+03; aff1C[473, 1] := 4.30447E-02;
aff1C[474, 0] := 4.74052E+03; aff1C[474, 1] := 4.28909E-02;
aff1C[475, 0] := 4.75050E+03; aff1C[475, 1] := 4.27380E-02;
aff1C[476, 0] := 4.76048E+03; aff1C[476, 1] := 4.25858E-02;
aff1C[477, 0] := 4.77046E+03; aff1C[477, 1] := 4.24345E-02;
aff1C[478, 0] := 4.78044E+03; aff1C[478, 1] := 4.22839E-02;
aff1C[479, 0] := 4.79042E+03; aff1C[479, 1] := 4.21341E-02;
aff1C[480, 0] := 4.80040E+03; aff1C[480, 1] := 4.19851E-02;
aff1C[481, 0] := 4.81038E+03; aff1C[481, 1] := 4.18368E-02;
aff1C[482, 0] := 4.82036E+03; aff1C[482, 1] := 4.16893E-02;
aff1C[483, 0] := 4.83034E+03; aff1C[483, 1] := 4.15425E-02;
aff1C[484, 0] := 4.84032E+03; aff1C[484, 1] := 4.13965E-02;
aff1C[485, 0] := 4.85030E+03; aff1C[485, 1] := 4.12512E-02;
aff1C[486, 0] := 4.86028E+03; aff1C[486, 1] := 4.11067E-02;
aff1C[487, 0] := 4.87026E+03; aff1C[487, 1] := 4.09629E-02;
aff1C[488, 0] := 4.88024E+03; aff1C[488, 1] := 4.08199E-02;
aff1C[489, 0] := 4.89022E+03; aff1C[489, 1] := 4.06776E-02;
aff1C[490, 0] := 4.90020E+03; aff1C[490, 1] := 4.05360E-02;
aff1C[491, 0] := 4.91018E+03; aff1C[491, 1] := 4.03951E-02;
aff1C[492, 0] := 4.92016E+03; aff1C[492, 1] := 4.02549E-02;
aff1C[493, 0] := 4.93014E+03; aff1C[493, 1] := 4.01154E-02;
aff1C[494, 0] := 4.94012E+03; aff1C[494, 1] := 3.99767E-02;
aff1C[495, 0] := 4.95010E+03; aff1C[495, 1] := 3.98386E-02;
aff1C[496, 0] := 4.96008E+03; aff1C[496, 1] := 3.97012E-02;
aff1C[497, 0] := 4.97006E+03; aff1C[497, 1] := 3.95645E-02;
aff1C[498, 0] := 4.98004E+03; aff1C[498, 1] := 3.94285E-02;
aff1C[499, 0] := 4.99002E+03; aff1C[499, 1] := 3.92932E-02;
aff1C[500, 0] := 5.00000E+03; aff1C[500, 1] := 3.91586E-02;
aff1C[501, 0] := 5.05000E+03; aff1C[501, 1] := 3.84940E-02;
aff1C[502, 0] := 5.10000E+03; aff1C[502, 1] := 3.78458E-02;
aff1C[503, 0] := 5.15000E+03; aff1C[503, 1] := 3.72134E-02;
aff1C[504, 0] := 5.20000E+03; aff1C[504, 1] := 3.65963E-02;
aff1C[505, 0] := 5.25000E+03; aff1C[505, 1] := 3.59941E-02;
aff1C[506, 0] := 5.30000E+03; aff1C[506, 1] := 3.54063E-02;
aff1C[507, 0] := 5.35000E+03; aff1C[507, 1] := 3.48326E-02;
aff1C[508, 0] := 5.40000E+03; aff1C[508, 1] := 3.42717E-02;
aff1C[509, 0] := 5.45000E+03; aff1C[509, 1] := 3.37227E-02;
aff1C[510, 0] := 5.50000E+03; aff1C[510, 1] := 3.31852E-02;
aff1C[511, 0] := 5.55000E+03; aff1C[511, 1] := 3.26591E-02;
aff1C[512, 0] := 5.60000E+03; aff1C[512, 1] := 3.21441E-02;
aff1C[513, 0] := 5.65000E+03; aff1C[513, 1] := 3.16398E-02;
aff1C[514, 0] := 5.70000E+03; aff1C[514, 1] := 3.11460E-02;
aff1C[515, 0] := 5.75000E+03; aff1C[515, 1] := 3.06625E-02;
aff1C[516, 0] := 5.80000E+03; aff1C[516, 1] := 3.01890E-02;
aff1C[517, 0] := 5.85000E+03; aff1C[517, 1] := 2.97253E-02;
aff1C[518, 0] := 5.90000E+03; aff1C[518, 1] := 2.92711E-02;
aff1C[519, 0] := 5.95000E+03; aff1C[519, 1] := 2.88261E-02;
aff1C[520, 0] := 6.00000E+03; aff1C[520, 1] := 2.83901E-02;
aff1C[521, 0] := 6.05000E+03; aff1C[521, 1] := 2.79630E-02;
aff1C[522, 0] := 6.10000E+03; aff1C[522, 1] := 2.75444E-02;
aff1C[523, 0] := 6.15000E+03; aff1C[523, 1] := 2.71342E-02;
aff1C[524, 0] := 6.20000E+03; aff1C[524, 1] := 2.67321E-02;
aff1C[525, 0] := 6.25000E+03; aff1C[525, 1] := 2.63380E-02;
aff1C[526, 0] := 6.30000E+03; aff1C[526, 1] := 2.59516E-02;
aff1C[527, 0] := 6.35000E+03; aff1C[527, 1] := 2.55727E-02;
aff1C[528, 0] := 6.40000E+03; aff1C[528, 1] := 2.52012E-02;
aff1C[529, 0] := 6.45000E+03; aff1C[529, 1] := 2.48369E-02;
aff1C[530, 0] := 6.50000E+03; aff1C[530, 1] := 2.44796E-02;
aff1C[531, 0] := 6.55000E+03; aff1C[531, 1] := 2.41291E-02;
aff1C[532, 0] := 6.60000E+03; aff1C[532, 1] := 2.37853E-02;
aff1C[533, 0] := 6.65000E+03; aff1C[533, 1] := 2.34479E-02;
aff1C[534, 0] := 6.70000E+03; aff1C[534, 1] := 2.31169E-02;
aff1C[535, 0] := 6.75000E+03; aff1C[535, 1] := 2.27920E-02;
aff1C[536, 0] := 6.80000E+03; aff1C[536, 1] := 2.24732E-02;
aff1C[537, 0] := 6.85000E+03; aff1C[537, 1] := 2.21602E-02;
aff1C[538, 0] := 6.90000E+03; aff1C[538, 1] := 2.18530E-02;
aff1C[539, 0] := 6.95000E+03; aff1C[539, 1] := 2.15514E-02;
aff1C[540, 0] := 7.00000E+03; aff1C[540, 1] := 2.12553E-02;
aff1C[541, 0] := 7.05000E+03; aff1C[541, 1] := 2.09645E-02;
aff1C[542, 0] := 7.10000E+03; aff1C[542, 1] := 2.06789E-02;
aff1C[543, 0] := 7.15000E+03; aff1C[543, 1] := 2.03983E-02;
aff1C[544, 0] := 7.20000E+03; aff1C[544, 1] := 2.01228E-02;
aff1C[545, 0] := 7.25000E+03; aff1C[545, 1] := 1.98521E-02;
aff1C[546, 0] := 7.30000E+03; aff1C[546, 1] := 1.95862E-02;
aff1C[547, 0] := 7.35000E+03; aff1C[547, 1] := 1.93248E-02;
aff1C[548, 0] := 7.40000E+03; aff1C[548, 1] := 1.90680E-02;
aff1C[549, 0] := 7.45000E+03; aff1C[549, 1] := 1.88156E-02;
aff1C[550, 0] := 7.50000E+03; aff1C[550, 1] := 1.85676E-02;
aff1C[551, 0] := 7.55000E+03; aff1C[551, 1] := 1.83237E-02;
aff1C[552, 0] := 7.60000E+03; aff1C[552, 1] := 1.80840E-02;
aff1C[553, 0] := 7.65000E+03; aff1C[553, 1] := 1.78484E-02;
aff1C[554, 0] := 7.70000E+03; aff1C[554, 1] := 1.76166E-02;
aff1C[555, 0] := 7.75000E+03; aff1C[555, 1] := 1.73888E-02;
aff1C[556, 0] := 7.80000E+03; aff1C[556, 1] := 1.71647E-02;
aff1C[557, 0] := 7.85000E+03; aff1C[557, 1] := 1.69442E-02;
aff1C[558, 0] := 7.90000E+03; aff1C[558, 1] := 1.67274E-02;
aff1C[559, 0] := 7.95000E+03; aff1C[559, 1] := 1.65142E-02;
aff1C[560, 0] := 8.00000E+03; aff1C[560, 1] := 1.63044E-02;
aff1C[561, 0] := 8.05000E+03; aff1C[561, 1] := 1.60979E-02;
aff1C[562, 0] := 8.10000E+03; aff1C[562, 1] := 1.58948E-02;
aff1C[563, 0] := 8.15000E+03; aff1C[563, 1] := 1.56949E-02;
aff1C[564, 0] := 8.20000E+03; aff1C[564, 1] := 1.54982E-02;
aff1C[565, 0] := 8.25000E+03; aff1C[565, 1] := 1.53046E-02;
aff1C[566, 0] := 8.30000E+03; aff1C[566, 1] := 1.51140E-02;
aff1C[567, 0] := 8.35000E+03; aff1C[567, 1] := 1.49264E-02;
aff1C[568, 0] := 8.40000E+03; aff1C[568, 1] := 1.47417E-02;
aff1C[569, 0] := 8.45000E+03; aff1C[569, 1] := 1.45599E-02;
aff1C[570, 0] := 8.50000E+03; aff1C[570, 1] := 1.43808E-02;
aff1C[571, 0] := 8.55000E+03; aff1C[571, 1] := 1.42045E-02;
aff1C[572, 0] := 8.60000E+03; aff1C[572, 1] := 1.40309E-02;
aff1C[573, 0] := 8.65000E+03; aff1C[573, 1] := 1.38599E-02;
aff1C[574, 0] := 8.70000E+03; aff1C[574, 1] := 1.36915E-02;
aff1C[575, 0] := 8.75000E+03; aff1C[575, 1] := 1.35256E-02;
aff1C[576, 0] := 8.80000E+03; aff1C[576, 1] := 1.33622E-02;
aff1C[577, 0] := 8.85000E+03; aff1C[577, 1] := 1.32009E-02;
aff1C[578, 0] := 8.90000E+03; aff1C[578, 1] := 1.30430E-02;
aff1C[579, 0] := 8.95000E+03; aff1C[579, 1] := 1.28911E-02;
aff1C[580, 0] := 9.00000E+03; aff1C[580, 1] := 1.27429E-02;
aff1C[581, 0] := 9.05000E+03; aff1C[581, 1] := 1.25956E-02;
aff1C[582, 0] := 9.10000E+03; aff1C[582, 1] := 1.24496E-02;
aff1C[583, 0] := 9.15000E+03; aff1C[583, 1] := 1.23055E-02;
aff1C[584, 0] := 9.20000E+03; aff1C[584, 1] := 1.21632E-02;
aff1C[585, 0] := 9.25000E+03; aff1C[585, 1] := 1.20225E-02;
aff1C[586, 0] := 9.30000E+03; aff1C[586, 1] := 1.18835E-02;
aff1C[587, 0] := 9.35000E+03; aff1C[587, 1] := 1.17461E-02;
aff1C[588, 0] := 9.40000E+03; aff1C[588, 1] := 1.16105E-02;
aff1C[589, 0] := 9.45000E+03; aff1C[589, 1] := 1.14765E-02;
aff1C[590, 0] := 9.50000E+03; aff1C[590, 1] := 1.13442E-02;
aff1C[591, 0] := 9.55000E+03; aff1C[591, 1] := 1.12135E-02;
aff1C[592, 0] := 9.60000E+03; aff1C[592, 1] := 1.10845E-02;
aff1C[593, 0] := 9.65000E+03; aff1C[593, 1] := 1.09571E-02;
aff1C[594, 0] := 9.70000E+03; aff1C[594, 1] := 1.08312E-02;
aff1C[595, 0] := 9.75000E+03; aff1C[595, 1] := 1.07069E-02;
aff1C[596, 0] := 9.80000E+03; aff1C[596, 1] := 1.05842E-02;
aff1C[597, 0] := 9.85000E+03; aff1C[597, 1] := 1.04630E-02;
aff1C[598, 0] := 9.90000E+03; aff1C[598, 1] := 1.03434E-02;
aff1C[599, 0] := 9.95000E+03; aff1C[599, 1] := 1.02252E-02;
aff1C[600, 0] := 1.00000E+04; aff1C[600, 1] := 1.01085E-02;
aff1C[601, 0] := 1.00500E+04; aff1C[601, 1] := 9.99326E-03;
aff1C[602, 0] := 1.01000E+04; aff1C[602, 1] := 9.87944E-03;
aff1C[603, 0] := 1.01500E+04; aff1C[603, 1] := 9.76705E-03;
aff1C[604, 0] := 1.02000E+04; aff1C[604, 1] := 9.65604E-03;
aff1C[605, 0] := 1.02500E+04; aff1C[605, 1] := 9.54641E-03;
aff1C[606, 0] := 1.03000E+04; aff1C[606, 1] := 9.43813E-03;
aff1C[607, 0] := 1.03500E+04; aff1C[607, 1] := 9.33119E-03;
aff1C[608, 0] := 1.04000E+04; aff1C[608, 1] := 9.22555E-03;
aff1C[609, 0] := 1.04500E+04; aff1C[609, 1] := 9.12120E-03;
aff1C[610, 0] := 1.05000E+04; aff1C[610, 1] := 9.01813E-03;
aff1C[611, 0] := 1.05500E+04; aff1C[611, 1] := 8.91631E-03;
aff1C[612, 0] := 1.06000E+04; aff1C[612, 1] := 8.81574E-03;
aff1C[613, 0] := 1.06500E+04; aff1C[613, 1] := 8.71637E-03;
aff1C[614, 0] := 1.07000E+04; aff1C[614, 1] := 8.61821E-03;
aff1C[615, 0] := 1.07500E+04; aff1C[615, 1] := 8.52123E-03;
aff1C[616, 0] := 1.08000E+04; aff1C[616, 1] := 8.42541E-03;
aff1C[617, 0] := 1.08500E+04; aff1C[617, 1] := 8.33074E-03;
aff1C[618, 0] := 1.09000E+04; aff1C[618, 1] := 8.23719E-03;
aff1C[619, 0] := 1.09500E+04; aff1C[619, 1] := 8.14476E-03;
aff1C[620, 0] := 1.10000E+04; aff1C[620, 1] := 8.05342E-03;
aff1C[621, 0] := 1.10500E+04; aff1C[621, 1] := 7.96316E-03;
aff1C[622, 0] := 1.11000E+04; aff1C[622, 1] := 7.87395E-03;
aff1C[623, 0] := 1.11500E+04; aff1C[623, 1] := 7.78579E-03;
aff1C[624, 0] := 1.12000E+04; aff1C[624, 1] := 7.69866E-03;
aff1C[625, 0] := 1.12500E+04; aff1C[625, 1] := 7.61255E-03;
aff1C[626, 0] := 1.13000E+04; aff1C[626, 1] := 7.52743E-03;
aff1C[627, 0] := 1.13500E+04; aff1C[627, 1] := 7.44330E-03;
aff1C[628, 0] := 1.14000E+04; aff1C[628, 1] := 7.36014E-03;
aff1C[629, 0] := 1.14500E+04; aff1C[629, 1] := 7.27793E-03;
aff1C[630, 0] := 1.15000E+04; aff1C[630, 1] := 7.19666E-03;
aff1C[631, 0] := 1.15500E+04; aff1C[631, 1] := 7.11632E-03;
aff1C[632, 0] := 1.16000E+04; aff1C[632, 1] := 7.03689E-03;
aff1C[633, 0] := 1.16500E+04; aff1C[633, 1] := 6.95837E-03;
aff1C[634, 0] := 1.17000E+04; aff1C[634, 1] := 6.88072E-03;
aff1C[635, 0] := 1.17500E+04; aff1C[635, 1] := 6.80395E-03;
aff1C[636, 0] := 1.18000E+04; aff1C[636, 1] := 6.72804E-03;
aff1C[637, 0] := 1.18500E+04; aff1C[637, 1] := 6.65297E-03;
aff1C[638, 0] := 1.19000E+04; aff1C[638, 1] := 6.57874E-03;
aff1C[639, 0] := 1.19500E+04; aff1C[639, 1] := 6.50534E-03;
aff1C[640, 0] := 1.20000E+04; aff1C[640, 1] := 6.43275E-03;
aff1C[641, 0] := 1.20500E+04; aff1C[641, 1] := 6.36095E-03;
aff1C[642, 0] := 1.21000E+04; aff1C[642, 1] := 6.28995E-03;
aff1C[643, 0] := 1.21500E+04; aff1C[643, 1] := 6.21971E-03;
aff1C[644, 0] := 1.22000E+04; aff1C[644, 1] := 6.15024E-03;
aff1C[645, 0] := 1.22500E+04; aff1C[645, 1] := 6.08153E-03;
aff1C[646, 0] := 1.23000E+04; aff1C[646, 1] := 6.01356E-03;
aff1C[647, 0] := 1.23500E+04; aff1C[647, 1] := 5.94633E-03;
aff1C[648, 0] := 1.24000E+04; aff1C[648, 1] := 5.87981E-03;
aff1C[649, 0] := 1.24500E+04; aff1C[649, 1] := 5.81400E-03;
aff1C[650, 0] := 1.25000E+04; aff1C[650, 1] := 5.74890E-03;
aff1C[651, 0] := 1.25500E+04; aff1C[651, 1] := 5.68449E-03;
aff1C[652, 0] := 1.26000E+04; aff1C[652, 1] := 5.62076E-03;
aff1C[653, 0] := 1.26500E+04; aff1C[653, 1] := 5.55771E-03;
aff1C[654, 0] := 1.27000E+04; aff1C[654, 1] := 5.49532E-03;
aff1C[655, 0] := 1.27500E+04; aff1C[655, 1] := 5.43358E-03;
aff1C[656, 0] := 1.28000E+04; aff1C[656, 1] := 5.37249E-03;
aff1C[657, 0] := 1.28500E+04; aff1C[657, 1] := 5.31204E-03;
aff1C[658, 0] := 1.29000E+04; aff1C[658, 1] := 5.25221E-03;
aff1C[659, 0] := 1.29500E+04; aff1C[659, 1] := 5.19300E-03;
aff1C[660, 0] := 1.30000E+04; aff1C[660, 1] := 5.13440E-03;
aff1C[661, 0] := 1.30500E+04; aff1C[661, 1] := 5.07640E-03;
aff1C[662, 0] := 1.31000E+04; aff1C[662, 1] := 5.01900E-03;
aff1C[663, 0] := 1.31500E+04; aff1C[663, 1] := 4.96218E-03;
aff1C[664, 0] := 1.32000E+04; aff1C[664, 1] := 4.90594E-03;
aff1C[665, 0] := 1.32500E+04; aff1C[665, 1] := 4.85027E-03;
aff1C[666, 0] := 1.33000E+04; aff1C[666, 1] := 4.79516E-03;
aff1C[667, 0] := 1.33500E+04; aff1C[667, 1] := 4.74061E-03;
aff1C[668, 0] := 1.34000E+04; aff1C[668, 1] := 4.68660E-03;
aff1C[669, 0] := 1.34500E+04; aff1C[669, 1] := 4.63314E-03;
aff1C[670, 0] := 1.35000E+04; aff1C[670, 1] := 4.58021E-03;
aff1C[671, 0] := 1.35500E+04; aff1C[671, 1] := 4.52780E-03;
aff1C[672, 0] := 1.36000E+04; aff1C[672, 1] := 4.47591E-03;
aff1C[673, 0] := 1.36500E+04; aff1C[673, 1] := 4.42454E-03;
aff1C[674, 0] := 1.37000E+04; aff1C[674, 1] := 4.37367E-03;
aff1C[675, 0] := 1.37500E+04; aff1C[675, 1] := 4.32329E-03;
aff1C[676, 0] := 1.38000E+04; aff1C[676, 1] := 4.27341E-03;
aff1C[677, 0] := 1.38500E+04; aff1C[677, 1] := 4.22401E-03;
aff1C[678, 0] := 1.39000E+04; aff1C[678, 1] := 4.17510E-03;
aff1C[679, 0] := 1.39500E+04; aff1C[679, 1] := 4.12665E-03;
aff1C[680, 0] := 1.40000E+04; aff1C[680, 1] := 4.07868E-03;
aff1C[681, 0] := 1.40500E+04; aff1C[681, 1] := 4.03116E-03;
aff1C[682, 0] := 1.41000E+04; aff1C[682, 1] := 3.98411E-03;
aff1C[683, 0] := 1.41500E+04; aff1C[683, 1] := 3.93750E-03;
aff1C[684, 0] := 1.42000E+04; aff1C[684, 1] := 3.89134E-03;
aff1C[685, 0] := 1.42500E+04; aff1C[685, 1] := 3.84561E-03;
aff1C[686, 0] := 1.43000E+04; aff1C[686, 1] := 3.80031E-03;
aff1C[687, 0] := 1.43500E+04; aff1C[687, 1] := 3.75544E-03;
aff1C[688, 0] := 1.44000E+04; aff1C[688, 1] := 3.71099E-03;
aff1C[689, 0] := 1.44500E+04; aff1C[689, 1] := 3.66696E-03;
aff1C[690, 0] := 1.45000E+04; aff1C[690, 1] := 3.62335E-03;
aff1C[691, 0] := 1.45500E+04; aff1C[691, 1] := 3.58014E-03;
aff1C[692, 0] := 1.46000E+04; aff1C[692, 1] := 3.53732E-03;
aff1C[693, 0] := 1.46500E+04; aff1C[693, 1] := 3.49491E-03;
aff1C[694, 0] := 1.47000E+04; aff1C[694, 1] := 3.45288E-03;
aff1C[695, 0] := 1.47500E+04; aff1C[695, 1] := 3.41125E-03;
aff1C[696, 0] := 1.48000E+04; aff1C[696, 1] := 3.36999E-03;
aff1C[697, 0] := 1.48500E+04; aff1C[697, 1] := 3.32911E-03;
aff1C[698, 0] := 1.49000E+04; aff1C[698, 1] := 3.28861E-03;
aff1C[699, 0] := 1.49500E+04; aff1C[699, 1] := 3.24847E-03;
aff1C[700, 0] := 1.50000E+04; aff1C[700, 1] := 3.20869E-03;
aff1C[701, 0] := 1.50500E+04; aff1C[701, 1] := 3.16928E-03;
aff1C[702, 0] := 1.51000E+04; aff1C[702, 1] := 3.13021E-03;
aff1C[703, 0] := 1.51500E+04; aff1C[703, 1] := 3.09150E-03;
aff1C[704, 0] := 1.52000E+04; aff1C[704, 1] := 3.05314E-03;
aff1C[705, 0] := 1.52500E+04; aff1C[705, 1] := 3.01512E-03;
aff1C[706, 0] := 1.53000E+04; aff1C[706, 1] := 2.97743E-03;
aff1C[707, 0] := 1.53500E+04; aff1C[707, 1] := 2.94008E-03;
aff1C[708, 0] := 1.54000E+04; aff1C[708, 1] := 2.90305E-03;
aff1C[709, 0] := 1.54500E+04; aff1C[709, 1] := 2.86636E-03;
aff1C[710, 0] := 1.55000E+04; aff1C[710, 1] := 2.82999E-03;
aff1C[711, 0] := 1.55500E+04; aff1C[711, 1] := 2.79393E-03;
aff1C[712, 0] := 1.56000E+04; aff1C[712, 1] := 2.75820E-03;
aff1C[713, 0] := 1.56500E+04; aff1C[713, 1] := 2.72277E-03;
aff1C[714, 0] := 1.57000E+04; aff1C[714, 1] := 2.68765E-03;
aff1C[715, 0] := 1.57500E+04; aff1C[715, 1] := 2.65283E-03;
aff1C[716, 0] := 1.58000E+04; aff1C[716, 1] := 2.61831E-03;
aff1C[717, 0] := 1.58500E+04; aff1C[717, 1] := 2.58409E-03;
aff1C[718, 0] := 1.59000E+04; aff1C[718, 1] := 2.55017E-03;
aff1C[719, 0] := 1.59500E+04; aff1C[719, 1] := 2.51653E-03;
aff1C[720, 0] := 1.60000E+04; aff1C[720, 1] := 2.48319E-03;
aff1C[721, 0] := 1.60500E+04; aff1C[721, 1] := 2.45012E-03;
aff1C[722, 0] := 1.61000E+04; aff1C[722, 1] := 2.41734E-03;
aff1C[723, 0] := 1.61500E+04; aff1C[723, 1] := 2.38483E-03;
aff1C[724, 0] := 1.62000E+04; aff1C[724, 1] := 2.35259E-03;
aff1C[725, 0] := 1.62500E+04; aff1C[725, 1] := 2.32063E-03;
aff1C[726, 0] := 1.63000E+04; aff1C[726, 1] := 2.28893E-03;
aff1C[727, 0] := 1.63500E+04; aff1C[727, 1] := 2.25750E-03;
aff1C[728, 0] := 1.64000E+04; aff1C[728, 1] := 2.22634E-03;
aff1C[729, 0] := 1.64500E+04; aff1C[729, 1] := 2.19543E-03;
aff1C[730, 0] := 1.65000E+04; aff1C[730, 1] := 2.16478E-03;
aff1C[731, 0] := 1.65500E+04; aff1C[731, 1] := 2.13438E-03;
aff1C[732, 0] := 1.66000E+04; aff1C[732, 1] := 2.10423E-03;
aff1C[733, 0] := 1.66500E+04; aff1C[733, 1] := 2.07433E-03;
aff1C[734, 0] := 1.67000E+04; aff1C[734, 1] := 2.04468E-03;
aff1C[735, 0] := 1.67500E+04; aff1C[735, 1] := 2.01526E-03;
aff1C[736, 0] := 1.68000E+04; aff1C[736, 1] := 1.98609E-03;
aff1C[737, 0] := 1.68500E+04; aff1C[737, 1] := 1.95715E-03;
aff1C[738, 0] := 1.69000E+04; aff1C[738, 1] := 1.92845E-03;
aff1C[739, 0] := 1.69500E+04; aff1C[739, 1] := 1.89998E-03;
aff1C[740, 0] := 1.70000E+04; aff1C[740, 1] := 1.87174E-03;
aff1C[741, 0] := 1.70500E+04; aff1C[741, 1] := 1.84372E-03;
aff1C[742, 0] := 1.71000E+04; aff1C[742, 1] := 1.81593E-03;
aff1C[743, 0] := 1.71500E+04; aff1C[743, 1] := 1.78836E-03;
aff1C[744, 0] := 1.72000E+04; aff1C[744, 1] := 1.76101E-03;
aff1C[745, 0] := 1.72500E+04; aff1C[745, 1] := 1.73388E-03;
aff1C[746, 0] := 1.73000E+04; aff1C[746, 1] := 1.70696E-03;
aff1C[747, 0] := 1.73500E+04; aff1C[747, 1] := 1.68026E-03;
aff1C[748, 0] := 1.74000E+04; aff1C[748, 1] := 1.65377E-03;
aff1C[749, 0] := 1.74500E+04; aff1C[749, 1] := 1.62748E-03;
aff1C[750, 0] := 1.75000E+04; aff1C[750, 1] := 1.60141E-03;
aff1C[751, 0] := 1.75500E+04; aff1C[751, 1] := 1.57553E-03;
aff1C[752, 0] := 1.76000E+04; aff1C[752, 1] := 1.54986E-03;
aff1C[753, 0] := 1.76500E+04; aff1C[753, 1] := 1.52439E-03;
aff1C[754, 0] := 1.77000E+04; aff1C[754, 1] := 1.49912E-03;
aff1C[755, 0] := 1.77500E+04; aff1C[755, 1] := 1.47404E-03;
aff1C[756, 0] := 1.78000E+04; aff1C[756, 1] := 1.44915E-03;
aff1C[757, 0] := 1.78500E+04; aff1C[757, 1] := 1.42446E-03;
aff1C[758, 0] := 1.79000E+04; aff1C[758, 1] := 1.39995E-03;
aff1C[759, 0] := 1.79500E+04; aff1C[759, 1] := 1.37564E-03;
aff1C[760, 0] := 1.80000E+04; aff1C[760, 1] := 1.35150E-03;
aff1C[761, 0] := 1.80500E+04; aff1C[761, 1] := 1.32756E-03;
aff1C[762, 0] := 1.81000E+04; aff1C[762, 1] := 1.30379E-03;
aff1C[763, 0] := 1.81500E+04; aff1C[763, 1] := 1.28021E-03;
aff1C[764, 0] := 1.82000E+04; aff1C[764, 1] := 1.25680E-03;
aff1C[765, 0] := 1.82500E+04; aff1C[765, 1] := 1.23357E-03;
aff1C[766, 0] := 1.83000E+04; aff1C[766, 1] := 1.21052E-03;
aff1C[767, 0] := 1.83500E+04; aff1C[767, 1] := 1.18764E-03;
aff1C[768, 0] := 1.84000E+04; aff1C[768, 1] := 1.16493E-03;
aff1C[769, 0] := 1.84500E+04; aff1C[769, 1] := 1.14238E-03;
aff1C[770, 0] := 1.85000E+04; aff1C[770, 1] := 1.12001E-03;
aff1C[771, 0] := 1.85500E+04; aff1C[771, 1] := 1.09780E-03;
aff1C[772, 0] := 1.86000E+04; aff1C[772, 1] := 1.07576E-03;
aff1C[773, 0] := 1.86500E+04; aff1C[773, 1] := 1.05387E-03;
aff1C[774, 0] := 1.87000E+04; aff1C[774, 1] := 1.03215E-03;
aff1C[775, 0] := 1.87500E+04; aff1C[775, 1] := 1.01059E-03;
aff1C[776, 0] := 1.88000E+04; aff1C[776, 1] := 9.89190E-04;
aff1C[777, 0] := 1.88500E+04; aff1C[777, 1] := 9.67946E-04;
aff1C[778, 0] := 1.89000E+04; aff1C[778, 1] := 9.46858E-04;
aff1C[779, 0] := 1.89500E+04; aff1C[779, 1] := 9.25923E-04;
aff1C[780, 0] := 1.90000E+04; aff1C[780, 1] := 9.05138E-04;
aff1C[781, 0] := 1.90500E+04; aff1C[781, 1] := 8.84501E-04;
aff1C[782, 0] := 1.91000E+04; aff1C[782, 1] := 8.64013E-04;
aff1C[783, 0] := 1.91500E+04; aff1C[783, 1] := 8.43672E-04;
aff1C[784, 0] := 1.92000E+04; aff1C[784, 1] := 8.23479E-04;
aff1C[785, 0] := 1.92500E+04; aff1C[785, 1] := 8.03431E-04;
aff1C[786, 0] := 1.93000E+04; aff1C[786, 1] := 7.83527E-04;
aff1C[787, 0] := 1.93500E+04; aff1C[787, 1] := 7.63766E-04;
aff1C[788, 0] := 1.94000E+04; aff1C[788, 1] := 7.44145E-04;
aff1C[789, 0] := 1.94500E+04; aff1C[789, 1] := 7.24663E-04;
aff1C[790, 0] := 1.95000E+04; aff1C[790, 1] := 7.05318E-04;
aff1C[791, 0] := 1.95500E+04; aff1C[791, 1] := 6.86111E-04;
aff1C[792, 0] := 1.96000E+04; aff1C[792, 1] := 6.67039E-04;
aff1C[793, 0] := 1.96500E+04; aff1C[793, 1] := 6.48102E-04;
aff1C[794, 0] := 1.97000E+04; aff1C[794, 1] := 6.29297E-04;
aff1C[795, 0] := 1.97500E+04; aff1C[795, 1] := 6.10623E-04;
aff1C[796, 0] := 1.98000E+04; aff1C[796, 1] := 5.92079E-04;
aff1C[797, 0] := 1.98500E+04; aff1C[797, 1] := 5.73663E-04;
aff1C[798, 0] := 1.99000E+04; aff1C[798, 1] := 5.55376E-04;
aff1C[799, 0] := 1.99500E+04; aff1C[799, 1] := 5.37215E-04;
aff1C[800, 0] := 2.00000E+04; aff1C[800, 1] := 5.19181E-04;
aff1C[801, 0] := 2.00500E+04; aff1C[801, 1] := 5.01272E-04;
aff1C[802, 0] := 2.01000E+04; aff1C[802, 1] := 4.83486E-04;
aff1C[803, 0] := 2.01500E+04; aff1C[803, 1] := 4.65821E-04;
aff1C[804, 0] := 2.02000E+04; aff1C[804, 1] := 4.48277E-04;
aff1C[805, 0] := 2.02500E+04; aff1C[805, 1] := 4.30853E-04;
aff1C[806, 0] := 2.03000E+04; aff1C[806, 1] := 4.13547E-04;
aff1C[807, 0] := 2.03500E+04; aff1C[807, 1] := 3.96360E-04;
aff1C[808, 0] := 2.04000E+04; aff1C[808, 1] := 3.79290E-04;
aff1C[809, 0] := 2.04500E+04; aff1C[809, 1] := 3.62337E-04;
aff1C[810, 0] := 2.05000E+04; aff1C[810, 1] := 3.45498E-04;
aff1C[811, 0] := 2.05500E+04; aff1C[811, 1] := 3.28771E-04;
aff1C[812, 0] := 2.06000E+04; aff1C[812, 1] := 3.12155E-04;
aff1C[813, 0] := 2.06500E+04; aff1C[813, 1] := 2.95649E-04;
aff1C[814, 0] := 2.07000E+04; aff1C[814, 1] := 2.79254E-04;
aff1C[815, 0] := 2.07500E+04; aff1C[815, 1] := 2.62969E-04;
aff1C[816, 0] := 2.08000E+04; aff1C[816, 1] := 2.46793E-04;
aff1C[817, 0] := 2.08500E+04; aff1C[817, 1] := 2.30726E-04;
aff1C[818, 0] := 2.09000E+04; aff1C[818, 1] := 2.14765E-04;
aff1C[819, 0] := 2.09500E+04; aff1C[819, 1] := 1.98910E-04;
aff1C[820, 0] := 2.10000E+04; aff1C[820, 1] := 1.83159E-04;
aff1C[821, 0] := 2.10500E+04; aff1C[821, 1] := 1.67511E-04;
aff1C[822, 0] := 2.11000E+04; aff1C[822, 1] := 1.51966E-04;
aff1C[823, 0] := 2.11500E+04; aff1C[823, 1] := 1.36523E-04;
aff1C[824, 0] := 2.12000E+04; aff1C[824, 1] := 1.21182E-04;
aff1C[825, 0] := 2.12500E+04; aff1C[825, 1] := 1.05942E-04;
aff1C[826, 0] := 2.13000E+04; aff1C[826, 1] := 9.08016E-05;
aff1C[827, 0] := 2.13500E+04; aff1C[827, 1] := 7.57589E-05;
aff1C[828, 0] := 2.14000E+04; aff1C[828, 1] := 6.08123E-05;
aff1C[829, 0] := 2.14500E+04; aff1C[829, 1] := 4.59608E-05;
aff1C[830, 0] := 2.15000E+04; aff1C[830, 1] := 3.12045E-05;
aff1C[831, 0] := 2.15500E+04; aff1C[831, 1] := 1.65434E-05;
aff1C[832, 0] := 2.16000E+04; aff1C[832, 1] := 1.97765E-06;
aff1C[833, 0] := 2.16500E+04; aff1C[833, 1] := -1.24926E-05;
aff1C[834, 0] := 2.17000E+04; aff1C[834, 1] := -2.68692E-05;
aff1C[835, 0] := 2.17500E+04; aff1C[835, 1] := -4.11539E-05;
aff1C[836, 0] := 2.18000E+04; aff1C[836, 1] := -5.53485E-05;
aff1C[837, 0] := 2.18500E+04; aff1C[837, 1] := -6.94549E-05;
aff1C[838, 0] := 2.19000E+04; aff1C[838, 1] := -8.34734E-05;
aff1C[839, 0] := 2.19500E+04; aff1C[839, 1] := -9.74039E-05;
aff1C[840, 0] := 2.20000E+04; aff1C[840, 1] := -1.11246E-04;
aff1C[841, 0] := 2.20500E+04; aff1C[841, 1] := -1.25000E-04;
aff1C[842, 0] := 2.21000E+04; aff1C[842, 1] := -1.38666E-04;
aff1C[843, 0] := 2.21500E+04; aff1C[843, 1] := -1.52246E-04;
aff1C[844, 0] := 2.22000E+04; aff1C[844, 1] := -1.65740E-04;
aff1C[845, 0] := 2.22500E+04; aff1C[845, 1] := -1.79150E-04;
aff1C[846, 0] := 2.23000E+04; aff1C[846, 1] := -1.92476E-04;
aff1C[847, 0] := 2.23500E+04; aff1C[847, 1] := -2.05719E-04;
aff1C[848, 0] := 2.24000E+04; aff1C[848, 1] := -2.18881E-04;
aff1C[849, 0] := 2.24500E+04; aff1C[849, 1] := -2.31962E-04;
aff1C[850, 0] := 2.25000E+04; aff1C[850, 1] := -2.44963E-04;
aff1C[851, 0] := 2.25500E+04; aff1C[851, 1] := -2.57885E-04;
aff1C[852, 0] := 2.26000E+04; aff1C[852, 1] := -2.70728E-04;
aff1C[853, 0] := 2.26500E+04; aff1C[853, 1] := -2.83492E-04;
aff1C[854, 0] := 2.27000E+04; aff1C[854, 1] := -2.96176E-04;
aff1C[855, 0] := 2.27500E+04; aff1C[855, 1] := -3.08782E-04;
aff1C[856, 0] := 2.28000E+04; aff1C[856, 1] := -3.21309E-04;
aff1C[857, 0] := 2.28500E+04; aff1C[857, 1] := -3.33760E-04;
aff1C[858, 0] := 2.29000E+04; aff1C[858, 1] := -3.46135E-04;
aff1C[859, 0] := 2.29500E+04; aff1C[859, 1] := -3.58436E-04;
aff1C[860, 0] := 2.30000E+04; aff1C[860, 1] := -3.70663E-04;
aff1C[861, 0] := 2.30500E+04; aff1C[861, 1] := -3.82817E-04;
aff1C[862, 0] := 2.31000E+04; aff1C[862, 1] := -3.94898E-04;
aff1C[863, 0] := 2.31500E+04; aff1C[863, 1] := -4.06907E-04;
aff1C[864, 0] := 2.32000E+04; aff1C[864, 1] := -4.18843E-04;
aff1C[865, 0] := 2.32500E+04; aff1C[865, 1] := -4.30707E-04;
aff1C[866, 0] := 2.33000E+04; aff1C[866, 1] := -4.42501E-04;
aff1C[867, 0] := 2.33500E+04; aff1C[867, 1] := -4.54224E-04;
aff1C[868, 0] := 2.34000E+04; aff1C[868, 1] := -4.65878E-04;
aff1C[869, 0] := 2.34500E+04; aff1C[869, 1] := -4.77463E-04;
aff1C[870, 0] := 2.35000E+04; aff1C[870, 1] := -4.88979E-04;
aff1C[871, 0] := 2.35500E+04; aff1C[871, 1] := -5.00428E-04;
aff1C[872, 0] := 2.36000E+04; aff1C[872, 1] := -5.11808E-04;
aff1C[873, 0] := 2.36500E+04; aff1C[873, 1] := -5.23122E-04;
aff1C[874, 0] := 2.37000E+04; aff1C[874, 1] := -5.34369E-04;
aff1C[875, 0] := 2.37500E+04; aff1C[875, 1] := -5.45549E-04;
aff1C[876, 0] := 2.38000E+04; aff1C[876, 1] := -5.56664E-04;
aff1C[877, 0] := 2.38500E+04; aff1C[877, 1] := -5.67715E-04;
aff1C[878, 0] := 2.39000E+04; aff1C[878, 1] := -5.78701E-04;
aff1C[879, 0] := 2.39500E+04; aff1C[879, 1] := -5.89623E-04;
aff1C[880, 0] := 2.40000E+04; aff1C[880, 1] := -6.00482E-04;
aff1C[881, 0] := 2.40500E+04; aff1C[881, 1] := -6.11277E-04;
aff1C[882, 0] := 2.41000E+04; aff1C[882, 1] := -6.22010E-04;
aff1C[883, 0] := 2.41500E+04; aff1C[883, 1] := -6.32681E-04;
aff1C[884, 0] := 2.42000E+04; aff1C[884, 1] := -6.43290E-04;
aff1C[885, 0] := 2.42500E+04; aff1C[885, 1] := -6.53838E-04;
aff1C[886, 0] := 2.43000E+04; aff1C[886, 1] := -6.64325E-04;
aff1C[887, 0] := 2.43500E+04; aff1C[887, 1] := -6.74752E-04;
aff1C[888, 0] := 2.44000E+04; aff1C[888, 1] := -6.85119E-04;
aff1C[889, 0] := 2.44500E+04; aff1C[889, 1] := -6.95427E-04;
aff1C[890, 0] := 2.45000E+04; aff1C[890, 1] := -7.05677E-04;
aff1C[891, 0] := 2.45500E+04; aff1C[891, 1] := -7.15868E-04;
aff1C[892, 0] := 2.46000E+04; aff1C[892, 1] := -7.26002E-04;
aff1C[893, 0] := 2.46500E+04; aff1C[893, 1] := -7.36079E-04;
aff1C[894, 0] := 2.47000E+04; aff1C[894, 1] := -7.46099E-04;
aff1C[895, 0] := 2.47500E+04; aff1C[895, 1] := -7.56063E-04;
aff1C[896, 0] := 2.48000E+04; aff1C[896, 1] := -7.65971E-04;
aff1C[897, 0] := 2.48500E+04; aff1C[897, 1] := -7.75823E-04;
aff1C[898, 0] := 2.49000E+04; aff1C[898, 1] := -7.85620E-04;
aff1C[899, 0] := 2.49500E+04; aff1C[899, 1] := -7.95362E-04;
aff1C[900, 0] := 2.50000E+04; aff1C[900, 1] := -8.05049E-04;
aff1C[901, 0] := 2.50500E+04; aff1C[901, 1] := -8.14682E-04;
aff1C[902, 0] := 2.51000E+04; aff1C[902, 1] := -8.24261E-04;
aff1C[903, 0] := 2.51500E+04; aff1C[903, 1] := -8.33786E-04;
aff1C[904, 0] := 2.52000E+04; aff1C[904, 1] := -8.43258E-04;
aff1C[905, 0] := 2.52500E+04; aff1C[905, 1] := -8.52678E-04;
aff1C[906, 0] := 2.53000E+04; aff1C[906, 1] := -8.62046E-04;
aff1C[907, 0] := 2.53500E+04; aff1C[907, 1] := -8.71364E-04;
aff1C[908, 0] := 2.54000E+04; aff1C[908, 1] := -8.80630E-04;
aff1C[909, 0] := 2.54500E+04; aff1C[909, 1] := -8.89847E-04;
aff1C[910, 0] := 2.55000E+04; aff1C[910, 1] := -8.99013E-04;
aff1C[911, 0] := 2.55500E+04; aff1C[911, 1] := -9.08129E-04;
aff1C[912, 0] := 2.56000E+04; aff1C[912, 1] := -9.17195E-04;
aff1C[913, 0] := 2.56500E+04; aff1C[913, 1] := -9.26211E-04;
aff1C[914, 0] := 2.57000E+04; aff1C[914, 1] := -9.35178E-04;
aff1C[915, 0] := 2.57500E+04; aff1C[915, 1] := -9.44095E-04;
aff1C[916, 0] := 2.58000E+04; aff1C[916, 1] := -9.52964E-04;
aff1C[917, 0] := 2.58500E+04; aff1C[917, 1] := -9.61785E-04;
aff1C[918, 0] := 2.59000E+04; aff1C[918, 1] := -9.70557E-04;
aff1C[919, 0] := 2.59500E+04; aff1C[919, 1] := -9.79282E-04;
aff1C[920, 0] := 2.60000E+04; aff1C[920, 1] := -9.87959E-04;
aff1C[921, 0] := 2.60500E+04; aff1C[921, 1] := -9.96591E-04;
aff1C[922, 0] := 2.61000E+04; aff1C[922, 1] := -1.00518E-03;
aff1C[923, 0] := 2.61500E+04; aff1C[923, 1] := -1.01371E-03;
aff1C[924, 0] := 2.62000E+04; aff1C[924, 1] := -1.02221E-03;
aff1C[925, 0] := 2.62500E+04; aff1C[925, 1] := -1.03066E-03;
aff1C[926, 0] := 2.63000E+04; aff1C[926, 1] := -1.03906E-03;
aff1C[927, 0] := 2.63500E+04; aff1C[927, 1] := -1.04743E-03;
aff1C[928, 0] := 2.64000E+04; aff1C[928, 1] := -1.05575E-03;
aff1C[929, 0] := 2.64500E+04; aff1C[929, 1] := -1.06403E-03;
aff1C[930, 0] := 2.65000E+04; aff1C[930, 1] := -1.07226E-03;
aff1C[931, 0] := 2.65500E+04; aff1C[931, 1] := -1.08045E-03;
aff1C[932, 0] := 2.66000E+04; aff1C[932, 1] := -1.08858E-03;
aff1C[933, 0] := 2.66500E+04; aff1C[933, 1] := -1.09665E-03;
aff1C[934, 0] := 2.67000E+04; aff1C[934, 1] := -1.10467E-03;
aff1C[935, 0] := 2.67500E+04; aff1C[935, 1] := -1.11264E-03;
aff1C[936, 0] := 2.68000E+04; aff1C[936, 1] := -1.12056E-03;
aff1C[937, 0] := 2.68500E+04; aff1C[937, 1] := -1.12843E-03;
aff1C[938, 0] := 2.69000E+04; aff1C[938, 1] := -1.13626E-03;
aff1C[939, 0] := 2.69500E+04; aff1C[939, 1] := -1.14405E-03;
aff1C[940, 0] := 2.70000E+04; aff1C[940, 1] := -1.15180E-03;
aff1C[941, 0] := 2.70500E+04; aff1C[941, 1] := -1.15951E-03;
aff1C[942, 0] := 2.71000E+04; aff1C[942, 1] := -1.16719E-03;
aff1C[943, 0] := 2.71500E+04; aff1C[943, 1] := -1.17482E-03;
aff1C[944, 0] := 2.72000E+04; aff1C[944, 1] := -1.18242E-03;
aff1C[945, 0] := 2.72500E+04; aff1C[945, 1] := -1.18999E-03;
aff1C[946, 0] := 2.73000E+04; aff1C[946, 1] := -1.19752E-03;
aff1C[947, 0] := 2.73500E+04; aff1C[947, 1] := -1.20501E-03;
aff1C[948, 0] := 2.74000E+04; aff1C[948, 1] := -1.21246E-03;
aff1C[949, 0] := 2.74500E+04; aff1C[949, 1] := -1.21988E-03;
aff1C[950, 0] := 2.75000E+04; aff1C[950, 1] := -1.22726E-03;
aff1C[951, 0] := 2.75500E+04; aff1C[951, 1] := -1.23460E-03;
aff1C[952, 0] := 2.76000E+04; aff1C[952, 1] := -1.24191E-03;
aff1C[953, 0] := 2.76500E+04; aff1C[953, 1] := -1.24918E-03;
aff1C[954, 0] := 2.77000E+04; aff1C[954, 1] := -1.25642E-03;
aff1C[955, 0] := 2.77500E+04; aff1C[955, 1] := -1.26362E-03;
aff1C[956, 0] := 2.78000E+04; aff1C[956, 1] := -1.27079E-03;
aff1C[957, 0] := 2.78500E+04; aff1C[957, 1] := -1.27792E-03;
aff1C[958, 0] := 2.79000E+04; aff1C[958, 1] := -1.28502E-03;
aff1C[959, 0] := 2.79500E+04; aff1C[959, 1] := -1.29208E-03;
aff1C[960, 0] := 2.80000E+04; aff1C[960, 1] := -1.29911E-03;
aff1C[961, 0] := 2.80500E+04; aff1C[961, 1] := -1.30610E-03;
aff1C[962, 0] := 2.81000E+04; aff1C[962, 1] := -1.31306E-03;
aff1C[963, 0] := 2.81500E+04; aff1C[963, 1] := -1.31999E-03;
aff1C[964, 0] := 2.82000E+04; aff1C[964, 1] := -1.32688E-03;
aff1C[965, 0] := 2.82500E+04; aff1C[965, 1] := -1.33374E-03;
aff1C[966, 0] := 2.83000E+04; aff1C[966, 1] := -1.34057E-03;
aff1C[967, 0] := 2.83500E+04; aff1C[967, 1] := -1.34736E-03;
aff1C[968, 0] := 2.84000E+04; aff1C[968, 1] := -1.35412E-03;
aff1C[969, 0] := 2.84500E+04; aff1C[969, 1] := -1.36085E-03;
aff1C[970, 0] := 2.85000E+04; aff1C[970, 1] := -1.36755E-03;
aff1C[971, 0] := 2.85500E+04; aff1C[971, 1] := -1.37422E-03;
aff1C[972, 0] := 2.86000E+04; aff1C[972, 1] := -1.38085E-03;
aff1C[973, 0] := 2.86500E+04; aff1C[973, 1] := -1.38745E-03;
aff1C[974, 0] := 2.87000E+04; aff1C[974, 1] := -1.39401E-03;
aff1C[975, 0] := 2.87500E+04; aff1C[975, 1] := -1.40055E-03;
aff1C[976, 0] := 2.88000E+04; aff1C[976, 1] := -1.40705E-03;
aff1C[977, 0] := 2.88500E+04; aff1C[977, 1] := -1.41353E-03;
aff1C[978, 0] := 2.89000E+04; aff1C[978, 1] := -1.41997E-03;
aff1C[979, 0] := 2.89500E+04; aff1C[979, 1] := -1.42639E-03;
aff1C[980, 0] := 2.90000E+04; aff1C[980, 1] := -1.43277E-03;
aff1C[981, 0] := 2.90500E+04; aff1C[981, 1] := -1.43912E-03;
aff1C[982, 0] := 2.91000E+04; aff1C[982, 1] := -1.44545E-03;
aff1C[983, 0] := 2.91500E+04; aff1C[983, 1] := -1.45174E-03;
aff1C[984, 0] := 2.92000E+04; aff1C[984, 1] := -1.45800E-03;
aff1C[985, 0] := 2.92500E+04; aff1C[985, 1] := -1.46424E-03;
aff1C[986, 0] := 2.93000E+04; aff1C[986, 1] := -1.47044E-03;
aff1C[987, 0] := 2.93500E+04; aff1C[987, 1] := -1.47662E-03;
aff1C[988, 0] := 2.94000E+04; aff1C[988, 1] := -1.48276E-03;
aff1C[989, 0] := 2.94500E+04; aff1C[989, 1] := -1.48888E-03;
aff1C[990, 0] := 2.95000E+04; aff1C[990, 1] := -1.49497E-03;
aff1C[991, 0] := 2.95500E+04; aff1C[991, 1] := -1.50103E-03;
aff1C[992, 0] := 2.96000E+04; aff1C[992, 1] := -1.50706E-03;
aff1C[993, 0] := 2.96500E+04; aff1C[993, 1] := -1.51307E-03;
aff1C[994, 0] := 2.97000E+04; aff1C[994, 1] := -1.51904E-03;
aff1C[995, 0] := 2.97500E+04; aff1C[995, 1] := -1.52499E-03;
aff1C[996, 0] := 2.98000E+04; aff1C[996, 1] := -1.53091E-03;
aff1C[997, 0] := 2.98500E+04; aff1C[997, 1] := -1.53680E-03;
aff1C[998, 0] := 2.99000E+04; aff1C[998, 1] := -1.54267E-03;
aff1C[999, 0] := 2.99500E+04; aff1C[999, 1] := -1.54851E-03;

// Element = Al

